// TwinCAT 3 PLC project HMI_Library
// Title: IBF_HMI
// Company: Industrial Brains B.V.
// ProjectVersion: 0.0.0.0
// Description: Basic HMI screens for use with Utilities and device libraries
// ProgramVersion: 3.1.4023.0
// libraries:
//   IBF_Device, * (Industrial Brains B.V.)
//   IBF_Utilities, * (Industrial Brains B.V.)
//   Tc2_Standard, * (Beckhoff Automation GmbH)
//   VisuDialogs, * (System)
//   VisuUserMgmt, * (System)
// project tree:
//   GVL/ E_BaseVisu.TcTLEO (not stored), GVL_HMI.TcGVL
//   HMIControl/ FB_HMIControl.TcPOU
//   IconsAndPictures/Backgrounds/PNG/ BackgroundImagePool_PNG.TcIPO (not stored)
//   IconsAndPictures/Backgrounds/SVG/ BackGroundImagePool_SVG.TcIPO (not stored)
//   IconsAndPictures/Buttons/ Buttons_SVG.TcIPO (not stored), Buttons_PNG.TcIPO (not stored)
//   IconsAndPictures/Logos/ LogoPool_PNG.TcIPO (not stored), LogoPool_SVG.TcIPO (not stored)
//   InputFunctions/ FB_HMILREALInput.TcPOU, FB_HMIInputBase.TcPOU
//   Screens/Backgrounds/ BackgroundNoButton.TcVIS, Background_SafetyAndSettings_SVG.TcVIS, BackgroundWithBorder.TcVIS
//   Screens/Base/ BaseScreen.TcVIS
//   Screens/EventsAndMessage/ BasicMessageScreen.TcVIS, Estop.TcVIS, MessageScreen.TcVIS (excluded from build)
//   Screens/Manual/DeviceScreens/ VisuAnalogOutControl.TcVIS, VisuAnalogAxisControl.TcVIS, VisuAnlogInputControl.TcVIS, VisuAxisControl.TcVIS, VisuCylinderControl.TcVIS, VisuDigitalInputControl.TcVIS, VisuDigitalOutControl.TcVIS, VisuEncoderInput.TcVIS, VisuKL5151Control.TcVIS, VisuKL15XXControl.TcVIS, VisuPushbuttonLightControl.TcVIS, VisuPWMControl.TcVIS, VisuDoublePWMControl.TcVIS, VisuUndefinedControl.TcVIS, VisuValveControl.TcVIS, VisuTwoVelocityAxisControl.TcVIS
//   Screens/Manual/ ManualButton_PNG.TcVIS, ManualControl.TcVIS, toManualButton.TcVIS
//   Screens/Parameter/ ParameterControl.TcVIS, ParButton_PNG.TcVIS
//   Screens/Startup Screen/ LogoScreen_PNG.TcVIS, LogoScreenBliss_PNG.TcVIS, LogoScreen_SVG.TcVIS, LogoScreenBlanc_SVG.TcVIS
//   Screens/State_PNG/ Idle_PNG.TcVIS, Manual_PNG.TcVIS, Parameter_PNG.TcVIS, Settings_PNG.TcVIS
//   Screens/State_SVG/ Manual.TcVIS, ParameterScreen.TcVIS, Settings.TcVIS, Idle.TcVIS
//   TextLists/ E_ComponentTypes.TcTLO, E_FaultTypes.TcTLO, E_Locations.TcTLO, E_MessageNumbers.TcTLO, E_ParameterNames.TcTLO, GlobalTextList.TcGTLO, TL_MessageDiscriptions.TcTLO
//   / VisualizationManager.TcVMO (not stored)

// ---- GVL/GVL_HMI.TcGVL
{attribute 'qualified_only'}
VAR_GLOBAL
	fbHMIControl	: FB_HMIControl ; // HMI control function
	bCmdSemiAuto	: BOOL ; // Show semi automatic screen
	bCmdAutomatic 	: BOOL ; // Show automatic screen
	eShownScreen 	: E_BaseVisu := E_BaseVisu.Idle ;
	bCmdSettings	: BOOL := FALSE ; // show settings screen
	bCmdParemeter	: BOOL := FALSE ; // Show paremeter screen
	bCmdManual		: BOOL := FALSE ; // Show manual screen
	bEstopActive	: BOOL ; // emergency stop is active
	sCmdEstopText	: STRING := 'SAFETY FAULT' ; // Emergency stop screen text 
	nStartVisu		: E_BaseVisu := E_BaseVisu.Idle ;
	nSelectedMessage : INT; 
END_VAR

// ---- HMIControl/FB_HMIControl.TcPOU
FUNCTION_BLOCK FB_HMIControl
VAR_INPUT 
END_VAR
VAR_OUTPUT
	bHideMessage	: BOOL ;
	bHideEStop 		: BOOL ;
	bHideBorders	: BOOL ;
	sEstopText		: STRING ;
	sOperatorMessage: STRING ;
END_VAR
VAR // HMI
END_VAR
VAR
	bWritePar  			: BOOL ; // write paremeters 
	bReadPar			: BOOL ; // Read paremeter file
	feWriteParemeter 	: F_TRIG ; // Falling edge trigger on leaving paremeter or manual screen

	reToSettings 		: R_TRIG ; // go to settings
	ePreviousScreen		: E_BaseVisu ; // previous screen
	
	bDisableSettings	: BOOL ; // disable settings button
END_VAR

SetScreen();
SetPopups();
ButtonEnable();

METHOD PRIVATE ButtonEnable : BOOL
VAR_INPUT
END_VAR
// Disable Buttons 
	bDisableSettings := GVL_HMI.eShownScreen = E_BaseVisu.Automatic ;
END_METHOD

METHOD PRIVATE SetPopups : BOOL
VAR_INPUT
END_VAR
// Set popup screens 
bHideEStop 			:= NOT GVL_HMI.bEstopActive ;
bHideMessage 		:= GVL_Message.bHideFaults ;
sOperatorMessage 	:= GVL_Message.sOPeratorMessage ;

GVL_HMI.bEstopActive := FALSE ;
END_METHOD

METHOD INTERNAL SetScreen : BOOL
VAR_INPUT
END_VAR
// Look for edges 
	reToSettings		( CLK := GVL_HMI.bCmdSettings );
	feWriteParemeter 	( CLK := GVL_HMI.bCmdParemeter OR GVL_HMI.bCmdManual );

// save previous screen 
IF reToSettings.Q  THEN 
	ePreviousScreen := GVL_HMI.eShownScreen ;
END_IF	
	
// Hide border control 
bHideBorders := FALSE ;

// Check active screen	
IF GVL_HMI.bCmdParemeter THEN 
	GVL_HMI.eShownScreen 	:= E_BaseVisu.Parameter ;
ELSIF GVL_HMI.bCmdManual THEN 
	GVL_HMI.eShownScreen 	:= E_BaseVisu.Manual;
ELSIF GVL_HMI.bCmdSettings THEN 
	GVL_HMI.eShownScreen 	:= E_BaseVisu.Settings ;
ELSIF NOT GVL_HMI.bCmdSettings AND GVL_HMI.eShownScreen = E_BaseVisu.Settings THEN 
	GVL_HMI.eShownScreen	:= ePreviousScreen ;
ELSIF gvl_HMI.bCmdSemiAuto THEN 
	GVL_HMI.eShownScreen 	:= E_BaseVisu.SemiAutomatic;
	gvl_HMI.bCmdSemiAuto	:= FALSE ; 
ELSIF gvl_HMI.bCmdAutomatic THEN 
	GVL_HMI.eShownScreen := E_BaseVisu.Automatic ;
	gvl_HMI.bCmdSemiAuto	:= FALSE ;
ELSE 
	GVL_HMI.eShownScreen := E_BaseVisu.Idle;
	bHideBorders := TRUE  ;	
END_IF

// Write parameters to file
IF feWriteParemeter.Q THEN
	bWritePar := TRUE ;
END_IF

IF bWritePar THEN 
	bWritePar R= GVL_Parameters.fbParameterHandler.CmdSavePar();
END_IF
END_METHOD

END_FUNCTION_BLOCK

// ---- InputFunctions/FB_HMILREALInput.TcPOU
FUNCTION_BLOCK PUBLIC FB_HMILREALInput EXTENDS FB_HMIInputBase // Analog value input from HMI
VAR_INPUT
	fInputFromHMI	: LREAL ;
END_VAR
VAR_OUTPUT
	fOutputToPLC	: LREAL ;
END_VAR
VAR
END_VAR

// call base function 
SUPER^();

// Set output to PLC
SetOutputToPLC();

METHOD PUBLIC SetOutputToPLC : BOOL
VAR_INPUT
END_VAR
IF bEnable THEN 
	fOutputToPLC := fInputFromHMI ;
END_IF
END_METHOD

END_FUNCTION_BLOCK

// ---- InputFunctions/FB_HMIInputBase.TcPOU
FUNCTION_BLOCK ABSTRACT FB_HMIInputBase //Base function for HMI inputs
VAR_INPUT
	bEnable : BOOL := TRUE ;
END_VAR
VAR_OUTPUT
	bInVisible			: BOOL := TRUE ; // input is visible (standard := NOT bEnable )
	bDeactivateInput	: BOOL := TRUE ; // input is enabled (Standard := bEnable)
END_VAR
VAR
END_VAR

SetHMIInstructions();

METHOD INTERNAL SetHMIInstructions : BOOL
VAR_INPUT
END_VAR
bInVisible 			:= NOT bEnable ;
bDeactivateInput	:= NOT bEnable ;
END_METHOD

METHOD ABSTRACT SetOutputToPLC : BOOL
VAR_INPUT
END_VAR
END_METHOD

END_FUNCTION_BLOCK

// ---- Screens/Backgrounds/BackgroundNoButton.TcVIS
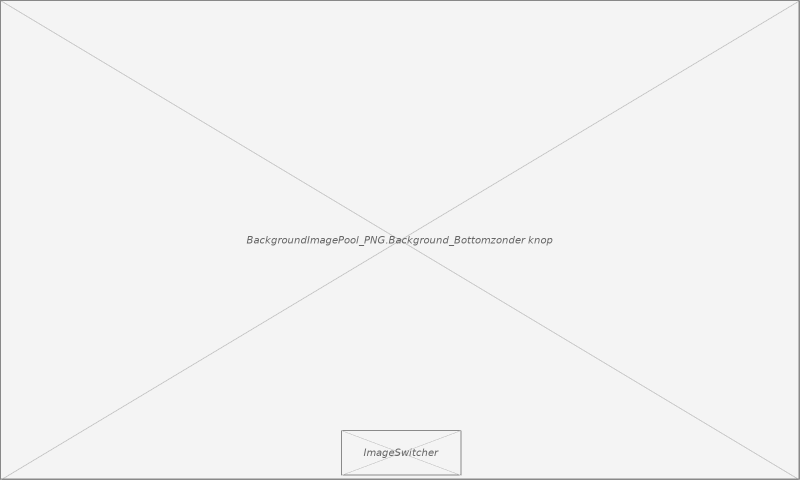
VISUALIZATION BackgroundNoButton  // 800x480
VAR_INPUT
	bHideEstop 			: BOOL ; // Hide emergency stop screen
	bDisableSettings	: BOOL ; // Deactivate settings
END_VAR
VAR_IN_OUT
	bCmdSettings	: BOOL ; // go to settings screen command
END_VAR
    Image (0,0 800x480), invisible if: bHideEstop, input disabled if: bHideEstop, image: BackgroundImagePool_PNG.Emergency Stop Active
    Image (0,0 800x480), image: BackgroundImagePool_PNG.Background_Bottomzonder knop
    ImageSwitcher (341,430 120x45), variable: GVL_HMI.bCmdSettings, input disabled if: bDisableSettings, background image: Buttons_PNG.Home-Settings Switch Pushed, image: Buttons_PNG.Home-Settings Switch, behaviour: TOGGLE
        p3148411668: Buttons_PNG.Home-Settings Switch Pushed
END_VISUALIZATION

// ---- Screens/Backgrounds/Background_SafetyAndSettings_SVG.TcVIS
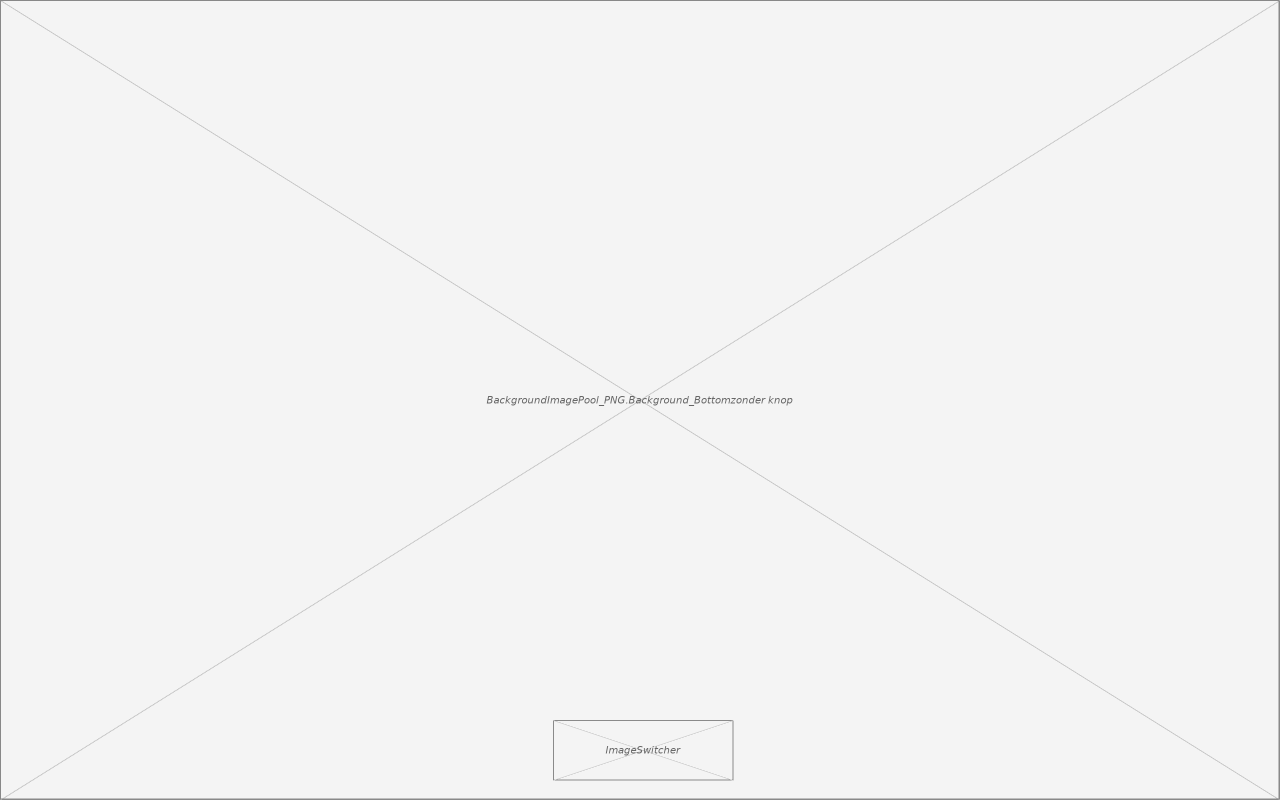
VISUALIZATION Background_SafetyAndSettings_SVG  // 1280x800
VAR_INPUT
	bHideEstop 			: BOOL ; // Hide emergency stop screen
	bDisableSettings	: BOOL ; // Deactivate settings
END_VAR
VAR_IN_OUT
	bCmdSettings	: BOOL ; // go to settings screen command
END_VAR
    Image (0,0 1280x800), invisible if: bHideEstop, input disabled if: bHideEstop, image: BackGroundImagePool_SVG.Emergency Stop Active 1280 x 800 Red Filled
    Image (0,0 1280x800), image: BackgroundImagePool_PNG.Background_Bottomzonder knop
    ImageSwitcher (553,720 180x60), variable: GVL_HMI.bCmdSettings, input disabled if: bDisableSettings, background image: Buttons_PNG.Home-Settings Switch Pushed, image: Buttons_PNG.Home-Settings Switch, behaviour: TOGGLE
        p3148411668: Buttons_PNG.Home-Settings Switch Pushed
END_VISUALIZATION

// ---- Screens/Backgrounds/BackgroundWithBorder.TcVIS
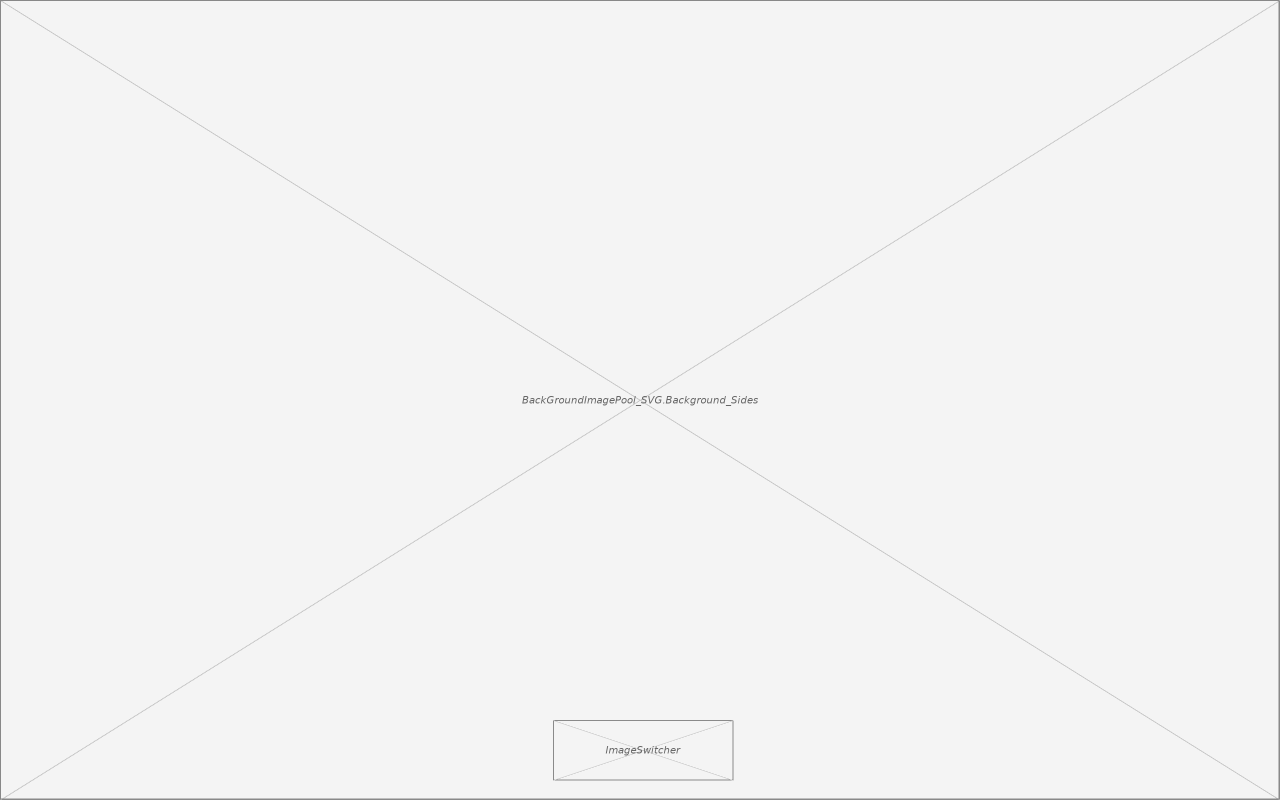
VISUALIZATION BackgroundWithBorder  // 1280x800
    Image (0,710 1280x90), image: BackGroundImagePool_SVG.Background_Bottom
    Image (0,0 1280x800), invisible if: GVL_HMI.fbHMIControl.bHideBorders, image: BackGroundImagePool_SVG.Background_Sides
    ImageSwitcher (553,720 180x60), variable: GVL_HMI.bCmdSettings, input disabled if: GVL_HMI.fbHMIControl.bDisableSettings, background image: Buttons_SVG.Home-Settings Switch Pushed, image: Buttons_SVG.Home Settings switch, behaviour: TOGGLE
        p3148411668: Buttons_SVG.Home-Settings Switch Pushed
END_VISUALIZATION

// ---- Screens/Base/BaseScreen.TcVIS
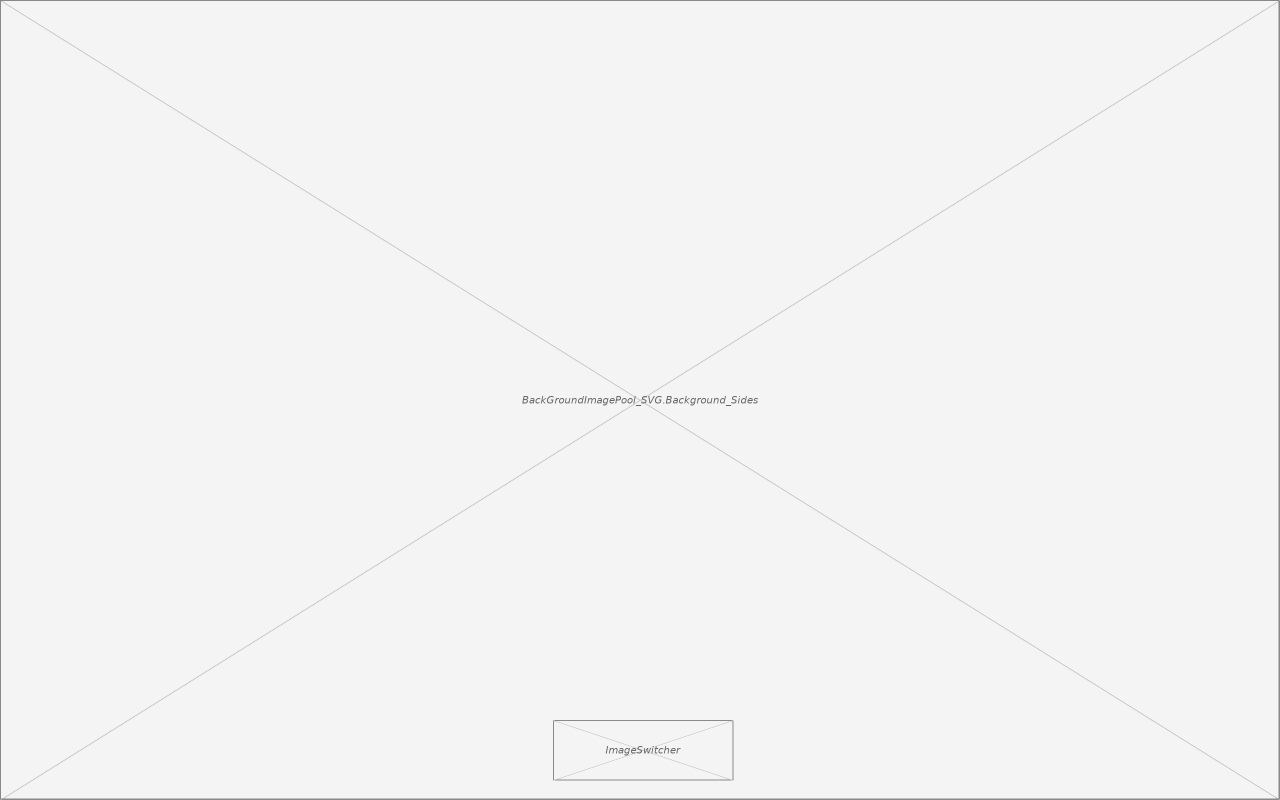
VISUALIZATION BaseScreen  // 1280x800
    Frame (0,0 1280x800)
        shows BackgroundWithBorder()
END_VISUALIZATION

// ---- Screens/EventsAndMessage/BasicMessageScreen.TcVIS
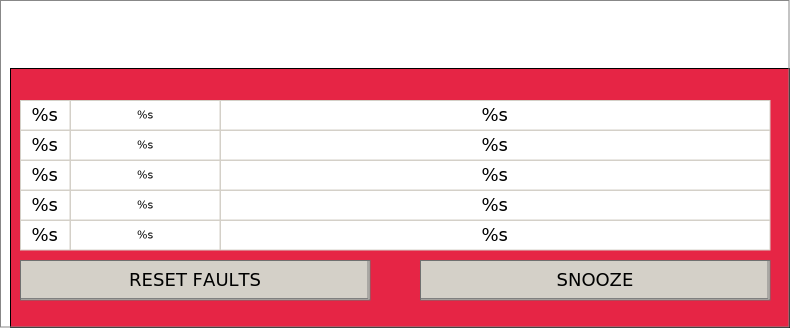
VISUALIZATION BasicMessageScreen  // 790x328
    RoundedRectangle (10,68 780x260)
    Group (20,100 754x200), invisible if: Utilities_Library.GVL_Message.bHideFaults, input disabled if: Utilities_Library.GVL_Message.bHideFaults
        Group (0,0 750x30)
            Textfield (0,0 50x30), "%s", text variable: GVL_Message.arActiveFaults[0].FaultType
            Textfield (50,0 150x30), "%s", text variable: Utilities_Library.GVL_Message.arActiveFaults[0].FullFaultId
            Textfield (200,0 550x30), "%s", text variable: Utilities_Library.GVL_Message.arActiveFaults[0].Discription
        Group (0,30 750x30)
            Textfield (0,0 50x30), "%s", text variable: Utilities_Library.GVL_Message.arActiveFaults[1].FaultType
            Textfield (50,0 150x30), "%s", text variable: Utilities_Library.GVL_Message.arActiveFaults[1].FullFaultId
            Textfield (200,0 550x30), "%s", text variable: Utilities_Library.GVL_Message.arActiveFaults[1].Discription
        Group (0,60 750x30)
            Textfield (0,0 50x30), "%s", text variable: Utilities_Library.GVL_Message.arActiveFaults[2].FaultType
            Textfield (50,0 150x30), "%s", text variable: Utilities_Library.GVL_Message.arActiveFaults[2].FullFaultId
            Textfield (200,0 550x30), "%s", text variable: Utilities_Library.GVL_Message.arActiveFaults[2].Discription
        Group (0,90 750x30)
            Textfield (0,0 50x30), "%s", text variable: Utilities_Library.GVL_Message.arActiveFaults[3].FaultType
            Textfield (50,0 150x30), "%s", text variable: Utilities_Library.GVL_Message.arActiveFaults[3].FullFaultId
            Textfield (200,0 550x30), "%s", text variable: Utilities_Library.GVL_Message.arActiveFaults[3].Discription
        Group (0,120 750x30)
            Textfield (0,0 50x30), "%s", text variable: Utilities_Library.GVL_Message.arActiveFaults[4].FaultType
            Textfield (50,0 150x30), "%s", text variable: Utilities_Library.GVL_Message.arActiveFaults[4].FullFaultId
            Textfield (200,0 550x30), "%s", text variable: Utilities_Library.GVL_Message.arActiveFaults[4].Discription
        Button (0,160 350x40), "RESET FAULTS", invisible if: Utilities_Library.GVL_Message.bHideReset, input disabled if: Utilities_Library.GVL_Message.bHideReset
            tap Utilities_Library.GVL_Message.bResetFaults
        Button (400,160 350x40), "SNOOZE"
            tap Utilities_Library.GVL_Message.bCmdSnoozeMessage
END_VISUALIZATION

// ---- Screens/EventsAndMessage/Estop.TcVIS
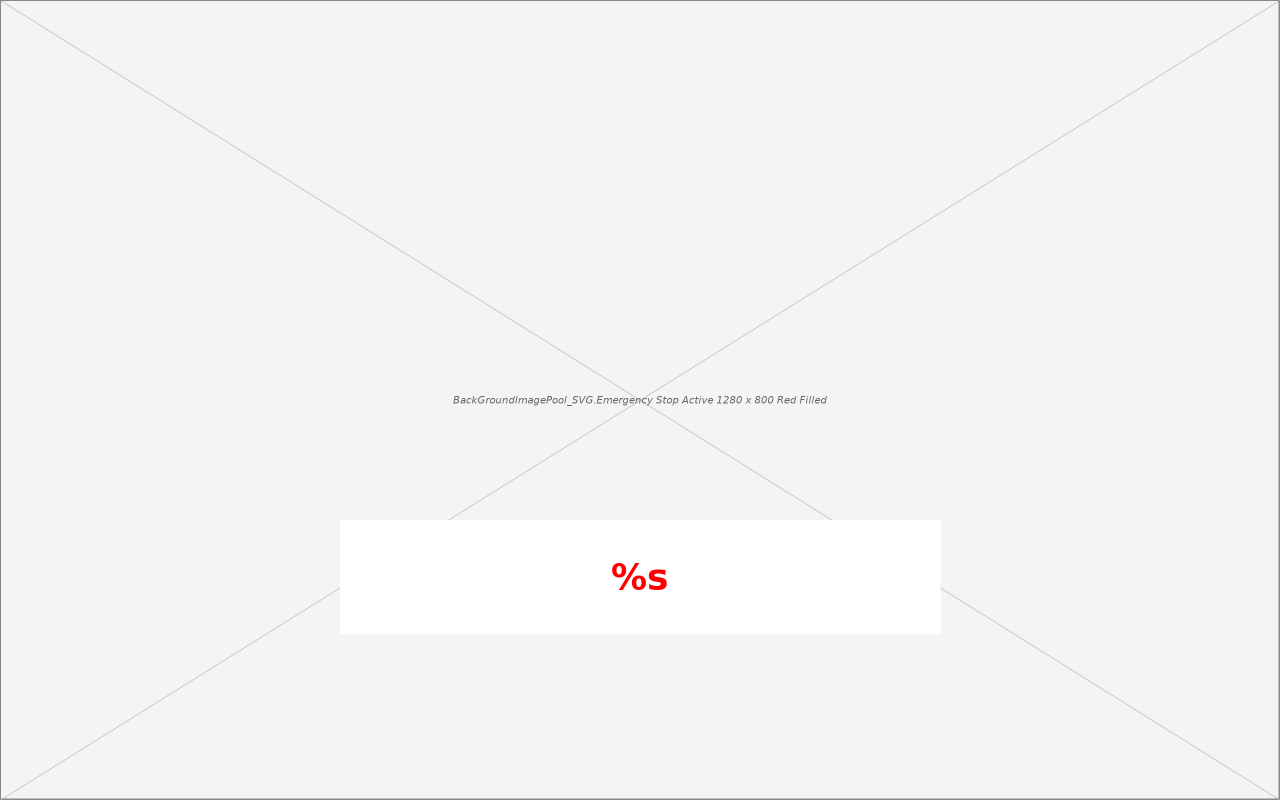
VISUALIZATION Estop  // 1280x800
VAR_IN_OUT
	bHideEstop		: BOOL ; // Hide Estop screen
END_VAR
    Image (0,0 1280x800), image: BackGroundImagePool_SVG.Emergency Stop Active 1280 x 800 Red Filled
    Textfield (340,520 600x114), "%s", text variable: GVL_HMI.sCmdEstopText
END_VISUALIZATION

// ---- Screens/Manual/DeviceScreens/VisuAnalogOutControl.TcVIS
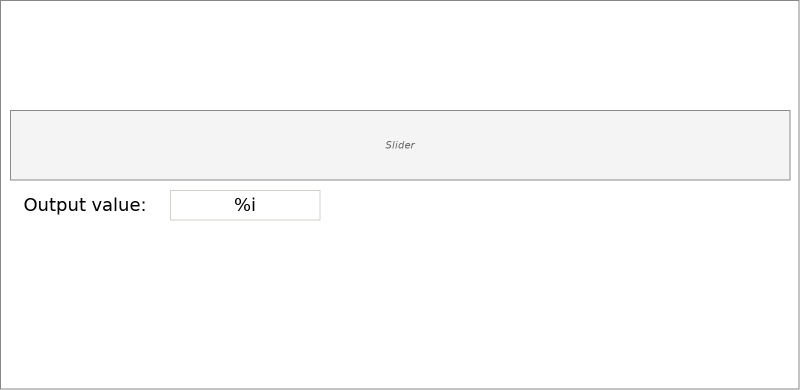
VISUALIZATION VisuAnalogOutControl  // 800x390
VAR_IN_OUT
	fbManualControler	: FB_ManualController ;
END_VAR
    Slider (10,110 780x70), variable: fbManualControler.pDevAnalogOut^.fCmdValue, scale 0..100
    Textfield (170,190 150x30), "%i", text variable: fbManualControler.pDevAnalogOut^.fCmdValue
        OnMouseClick: write the text variable via VisuDialogs.Numpad
    Label (10,190 150x30), "Output value:"
END_VISUALIZATION

// ---- Screens/Manual/DeviceScreens/VisuAnalogAxisControl.TcVIS
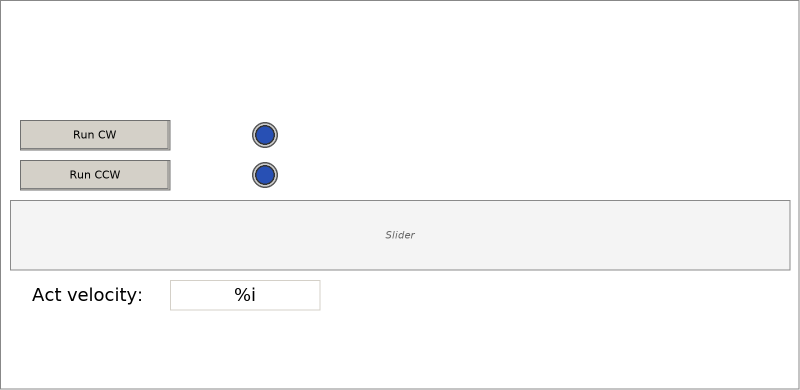
VISUALIZATION VisuAnalogAxisControl  // 800x390
VAR_IN_OUT
	fbManualControler	: FB_ManualController ;
END_VAR
    Slider (10,200 780x70), variable: fbManualControler.pDevAnalogAxis^.stManualCtrl.fCmdVelocity, scale 0..100
    Textfield (170,280 150x30), "%i", text variable: fbManualControler.pDevAnalogAxis^.fActVelocity
        OnMouseClick: write the text variable via VisuDialogs.Numpad
    Label (10,280 150x30), "Act velocity:"
    Button (20,120 150x30), "Run CW"
        tap fbManualControler.pDevAnalogAxis^.stManualCtrl.bCmdRunCW
    Button (20,160 150x30), "Run CCW"
        tap fbManualControler.pDevAnalogAxis^.stManualCtrl.bCmdRunCCW
    Lamp1 (190,120 150x30), variable: fbManualControler.pDevAnalogAxis^.bMovingCW, style: Lamp-Lamp1-Blue
    Lamp1 (190,160 150x30), variable: fbManualControler.pDevAnalogAxis^.bMovingCCW, style: Lamp-Lamp1-Blue
END_VISUALIZATION

// ---- Screens/Manual/DeviceScreens/VisuAnlogInputControl.TcVIS
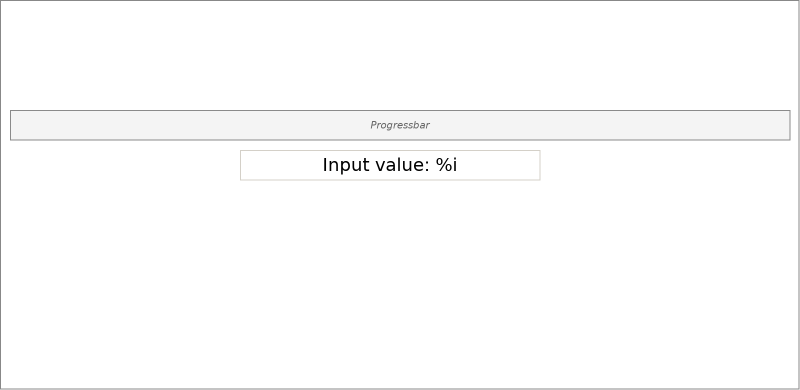
VISUALIZATION VisuAnlogInputControl  // 800x390
VAR_IN_OUT
	fbManualControler	: FB_ManualController ;
END_VAR
    Progressbar (10,110 780x30), variable: fbManualControler.pDevAnalogInput^.fValue
    Textfield (240,150 300x30), "Input value: %i", text variable: fbManualControler.pDevAnalogInput^.fValue
END_VISUALIZATION

// ---- Screens/Manual/DeviceScreens/VisuAxisControl.TcVIS
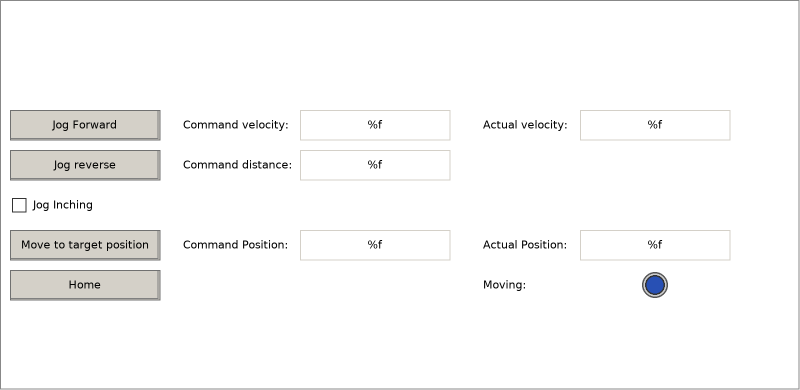
VISUALIZATION VisuAxisControl  // 800x390
VAR_IN_OUT
	fbManualControler	: FB_ManualController ;
END_VAR
    Button (10,110 150x30), "Jog Forward"
        tap fbManualControler.pDevAxis^.stManualCtrl.bCmdJogForward
    Button (10,150 150x30), "Jog reverse"
        tap fbManualControler.pDevAxis^.stManualCtrl.bCmdJogReverse
    Button (10,230 150x30), "Move to target position"
        tap fbManualControler.pDevAxis^.stManualCtrl.bCmdToPos
    Button (10,270 150x30), "Home"
        tap fbManualControler.pDevAxis^.stManualCtrl.bCmdHome
    Checkbox (10,190 150x30), "Jog Inching", variable: fbManualControler.pDevAxis^.stManualCtrl.bCmdInching
    Label (180,150 120x30), "Command distance:"
    Label (180,110 120x30), "Command velocity:"
    Label (180,230 120x30), "Command Position:"
    Textfield (300,110 150x30), "%f", text variable: fbManualControler.pDevAxis^.stManualCtrl.fVelocity
        OnMouseDown: write the text variable via VisuDialogs.Numpad
    Textfield (300,150 150x30), "%f", text variable: fbManualControler.pDevAxis^.stManualCtrl.fDistance
        OnMouseDown: write the text variable via VisuDialogs.Numpad
    Textfield (300,230 150x30), "%f", text variable: fbManualControler.pDevAxis^.stManualCtrl.fPosition
        OnMouseDown: write the text variable via VisuDialogs.Numpad
    Label (480,110 100x30), "Actual velocity:"
    Label (480,230 100x30), "Actual Position:"
    Textfield (580,230 150x30), "%f", text variable: fbManualControler.pDevAxis^.fActPosition
        OnMouseDown: write the text variable via VisuDialogs.Numpad
    Textfield (580,110 150x30), "%f", text variable: fbManualControler.pDevAxis^.fVelocity
        OnMouseDown: write the text variable via VisuDialogs.Numpad
    Lamp1 (580,270 150x30), variable: fbManualControler.pDevAxis^.AxisRef.Status.Moving, style: Lamp-Lamp1-Blue
    Label (480,270 100x30), "Moving:"
END_VISUALIZATION

// ---- Screens/Manual/DeviceScreens/VisuCylinderControl.TcVIS
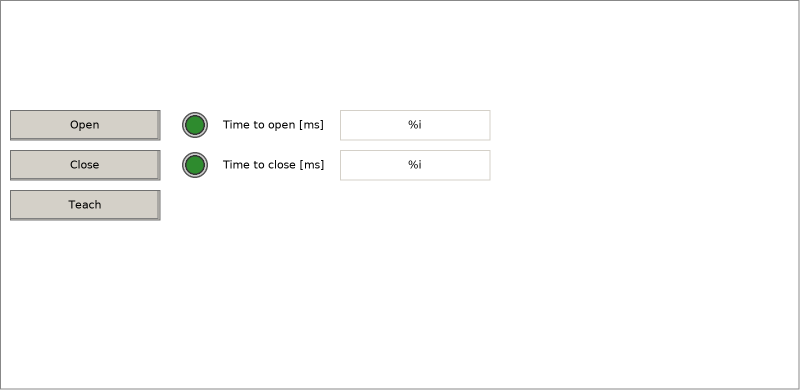
VISUALIZATION VisuCylinderControl  // 800x390
VAR_IN_OUT
	fbManualControler	: FB_ManualController ;
END_VAR
    Button (10,110 150x30), "Open"
        tap fbManualControler.pDevCylinder^.stManualCtrl.bCmdOpen
    Button (10,150 150x30), "Close"
        tap fbManualControler.pDevCylinder^.stManualCtrl.bCmdClose
    Lamp1 (180,110 30x30), variable: fbManualControler.pDevCylinder^.bFco_Open, style: Lamp-Lamp1-Green
    Button (10,190 150x30), "Teach"
        toggle fbManualControler.pDevCylinder^.stManualCtrl.bCmdTeach
    Lamp1 (180,150 30x30), variable: fbManualControler.pDevCylinder^.bFco_Closed, style: Lamp-Lamp1-Green
    Label (220,110 100x30), "Time to open [ms]"
    Label (220,150 100x30), "Time to close [ms]"
    Textfield (340,150 150x30), "%i", text variable: fbManualControler.pDevCylinder^.stParTimeToClose.fValue
        OnMouseClick: write the text variable via VisuDialogs.Numpad, min 0
    Textfield (340,110 150x30), "%i", text variable: fbManualControler.pDevCylinder^.stParTimeToOpen.fValue
        OnMouseClick: write the text variable via VisuDialogs.Numpad, min 0
END_VISUALIZATION

// ---- Screens/Manual/DeviceScreens/VisuDigitalInputControl.TcVIS
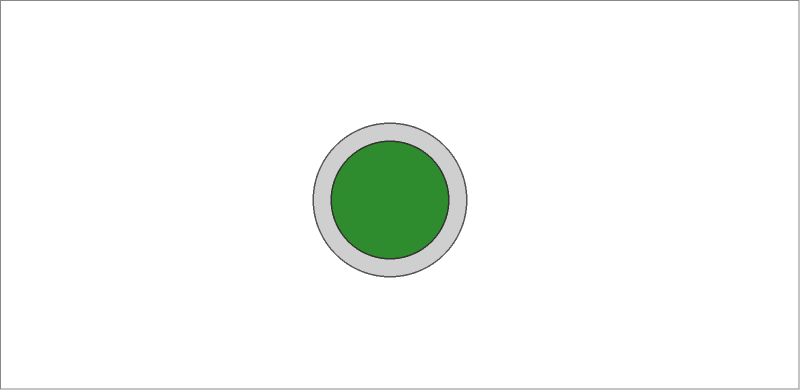
VISUALIZATION VisuDigitalInputControl  // 800x390
VAR_IN_OUT
	fbManualControler	: FB_ManualController ;
END_VAR
    Lamp1 (300,110 180x180), variable: fbManualControler.pDevDigitalInput^.bFcoInputActive, style: Lamp-Lamp1-Green
END_VISUALIZATION

// ---- Screens/Manual/DeviceScreens/VisuDigitalOutControl.TcVIS
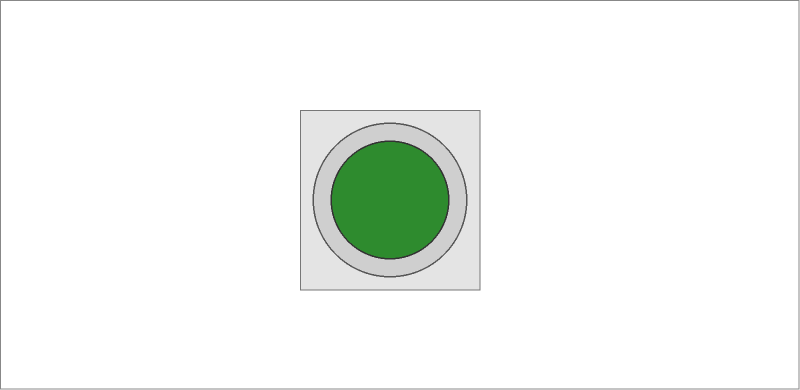
VISUALIZATION VisuDigitalOutControl  // 800x390
VAR_IN_OUT
	fbManualControler	: FB_ManualController ;
END_VAR
    PushSwitch (300,110 180x180), variable: fbManualControler.pDevDigitalOut^.bCmdOn, behaviour: TOGGLE, style: Switch-PushSwitch-Green
END_VISUALIZATION

// ---- Screens/Manual/DeviceScreens/VisuEncoderInput.TcVIS
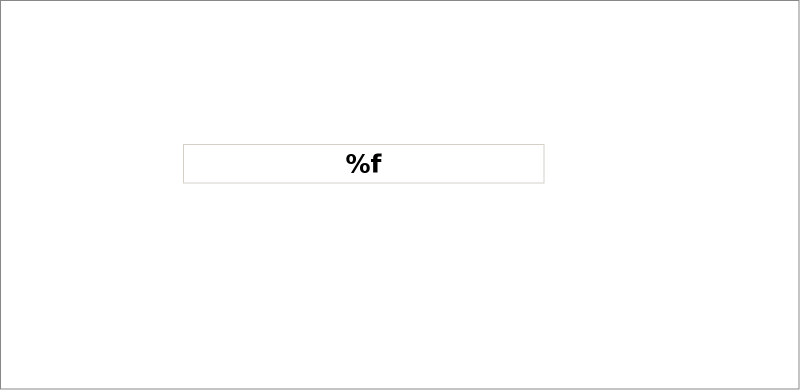
VISUALIZATION VisuEncoderInput  // 800x390
VAR_IN_OUT
	fbManualControler	: FB_ManualController ;
END_VAR
    Textfield (183,144 361x39), "%f", text variable: fbManualControler.pDevEncoder^.nOutPosition
END_VISUALIZATION

// ---- Screens/Manual/DeviceScreens/VisuKL5151Control.TcVIS
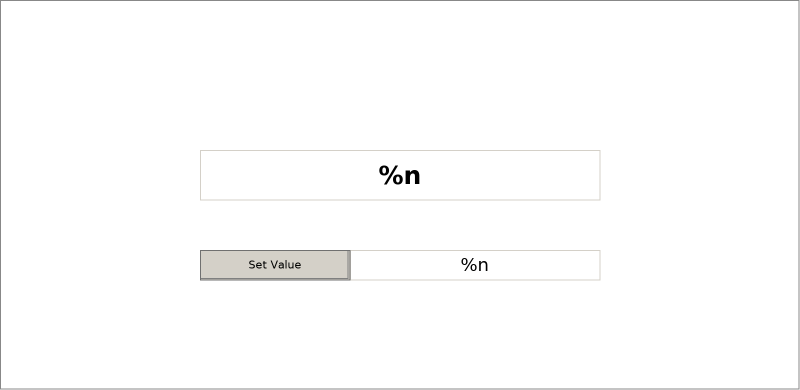
VISUALIZATION VisuKL5151Control  // 800x390
VAR_IN_OUT
	fbManualControler	: FB_ManualController ;
END_VAR
    Textfield (200,150 400x50), "%n", text variable: fbManualControler.pDevKL5151^.CountValue
    Textfield (350,250 250x30), "%n", text variable: fbManualControler.pDevKL5151^.stManualControl.nManValue
        OnMouseClick: write the text variable via VisuDialogs.Numpad
    Button (200,250 150x30), "Set Value"
        tap fbManualControler.pDevKL5151^.stManualControl.bManSetValue
END_VISUALIZATION

// ---- Screens/Manual/DeviceScreens/VisuKL15XXControl.TcVIS
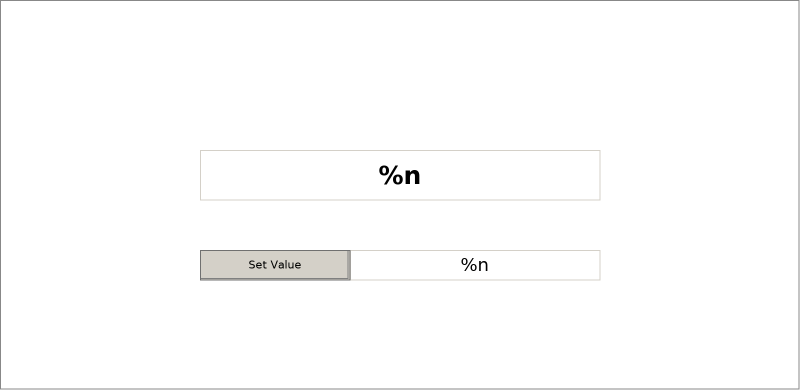
VISUALIZATION VisuKL15XXControl  // 800x390
VAR_IN_OUT
	fbManualControler	: FB_ManualController ;
END_VAR
    Textfield (200,150 400x50), "%n", text variable: fbManualControler.pDevKL1512^.CountValue
    Textfield (350,250 250x30), "%n", text variable: fbManualControler.pDevKL1512^.stManualControl.nManValue
        OnMouseClick: write the text variable via VisuDialogs.Numpad
    Button (200,250 150x30), "Set Value"
        tap fbManualControler.pDevKL1512^.stManualControl.bManSetValue
END_VISUALIZATION

// ---- Screens/Manual/DeviceScreens/VisuPushbuttonLightControl.TcVIS
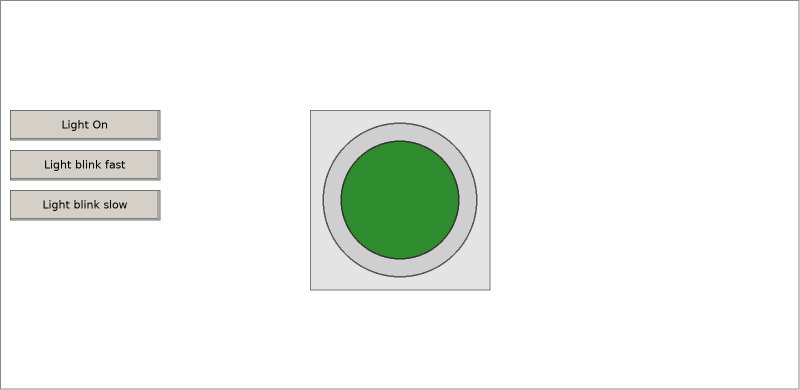
VISUALIZATION VisuPushbuttonLightControl  // 800x390
VAR_IN_OUT
	fbManualControler	: FB_ManualController ;
END_VAR
    PushSwitch (310,110 180x180), variable: fbManualControler.pDevPBL^.bFcoInputActive, behaviour: TOGGLE, style: Switch-PushSwitch-Green
    Button (10,110 150x30), "Light On"
        toggle fbManualControler.pDevPBL^.fbLight.bCmdOn
    Button (10,150 150x30), "Light blink fast"
        toggle fbManualControler.pDevPBL^.fbLight.bCmdBlinkFast
    Button (10,190 150x30), "Light blink slow"
        toggle fbManualControler.pDevPBL^.fbLight.bCmdBlinkSlow
END_VISUALIZATION

// ---- Screens/Manual/DeviceScreens/VisuPWMControl.TcVIS
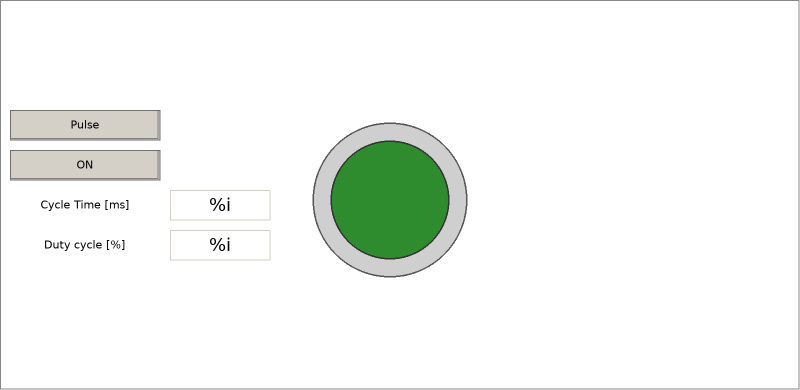
VISUALIZATION VisuPWMControl  // 800x390
VAR_IN_OUT
	fbManualControler	: FB_ManualController ;
END_VAR
    Lamp1 (300,110 180x180), variable: fbManualControler.pDevPWMController^.qbOutput, style: Lamp-Lamp1-Green
    Button (10,110 150x30), "Pulse"
        toggle fbManualControler.pDevPWMController^.bCmdPWMCycle
    Button (10,150 150x30), "ON"
        tap fbManualControler.pDevPWMController^.bCmdOn
    Textfield (170,190 100x30), "%i", text variable: fbManualControler.pDevPWMController^.nPeriodLength
        OnMouseUp: write the text variable via VisuDialogs.Numpad
    Label (10,190 150x30), "Cycle Time [ms]"
    Label (10,230 150x30), "Duty cycle [%]"
    Textfield (170,230 100x30), "%i", text variable: fbManualControler.pDevPWMController^.nDutyCycle
        OnMouseClick: write the text variable via VisuDialogs.Numpad, min 0, max 100
END_VISUALIZATION

// ---- Screens/Manual/DeviceScreens/VisuDoublePWMControl.TcVIS
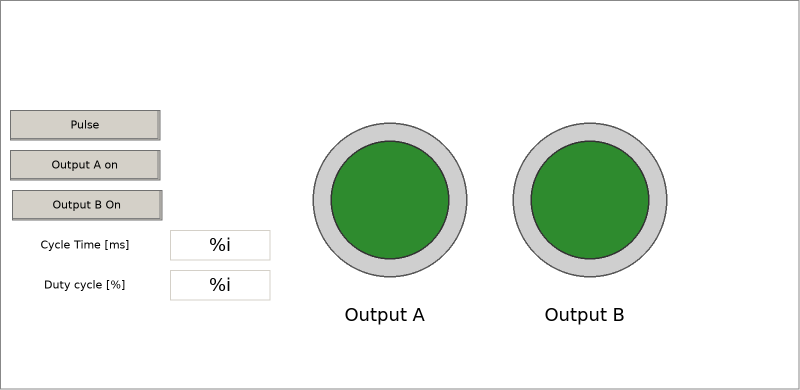
VISUALIZATION VisuDoublePWMControl  // 800x390
VAR_IN_OUT
	fbManualControler	: FB_ManualController ;
END_VAR
    Lamp1 (300,110 180x180), variable: fbManualControler.pDevDoublePWM^.qbOutputA, style: Lamp-Lamp1-Green
    Button (10,110 150x30), "Pulse"
        toggle fbManualControler.pDevDoublePWM^.bCmdPWMOn
    Button (10,150 150x30), "Output A on"
        toggle fbManualControler.pDevDoublePWM^.bCmdChanelAOn
    Textfield (170,230 100x30), "%i", text variable: fbManualControler.pDevDoublePWM^.stParPeriodLength.fValue
        OnMouseUp: write the text variable via VisuDialogs.Numpad
    Label (10,230 150x30), "Cycle Time [ms]"
    Label (10,270 150x30), "Duty cycle [%]"
    Textfield (170,270 100x30), "%i", text variable: fbManualControler.pDevDoublePWM^.stParDutyCycle.fValue
        OnMouseClick: write the text variable via VisuDialogs.Numpad, min 0, max 100
    Lamp1 (500,110 180x180), variable: fbManualControler.pDevPWMController^.qbOutput, style: Lamp-Lamp1-Green
    Button (12,190 150x30), "Output B On"
        tap fbManualControler.pDevDoublePWM^.bCmdChanelBOn
    Label (310,300 150x30), "Output A"
    Label (510,300 150x30), "Output B"
END_VISUALIZATION

// ---- Screens/Manual/DeviceScreens/VisuUndefinedControl.TcVIS
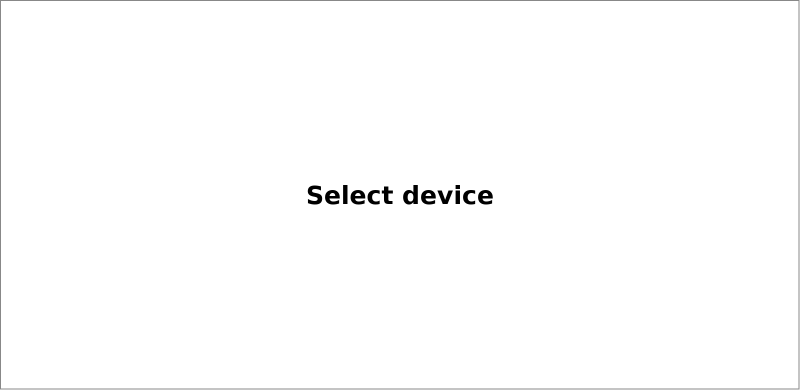
VISUALIZATION VisuUndefinedControl  // 800x390
    Label (0,0 800x390), "Select device"
END_VISUALIZATION

// ---- Screens/Manual/DeviceScreens/VisuValveControl.TcVIS
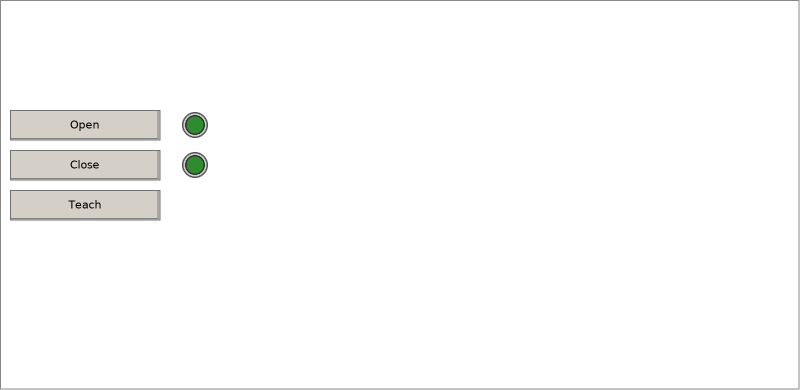
VISUALIZATION VisuValveControl  // 800x390
VAR_IN_OUT
	fbManualControler	: FB_ManualController ;
END_VAR
    Button (10,110 150x30), "Open"
        tap fbManualControler.pDevValve^.stManualCtrl.bCmdOpen
    Button (10,150 150x30), "Close"
        tap fbManualControler.pDevValve^.stManualCtrl.bCmdClose
    Lamp1 (180,110 30x30), variable: fbManualControler.pDevValve^.bFco_Open, style: Lamp-Lamp1-Green
    Button (10,190 150x30), "Teach"
        toggle fbManualControler.pDevValve^.stManualCtrl.bCmdTeach
    Lamp1 (180,150 30x30), variable: fbManualControler.pDevValve^.bFco_Closed, style: Lamp-Lamp1-Green
END_VISUALIZATION

// ---- Screens/EventsAndMessage/MessageScreen.TcVIS
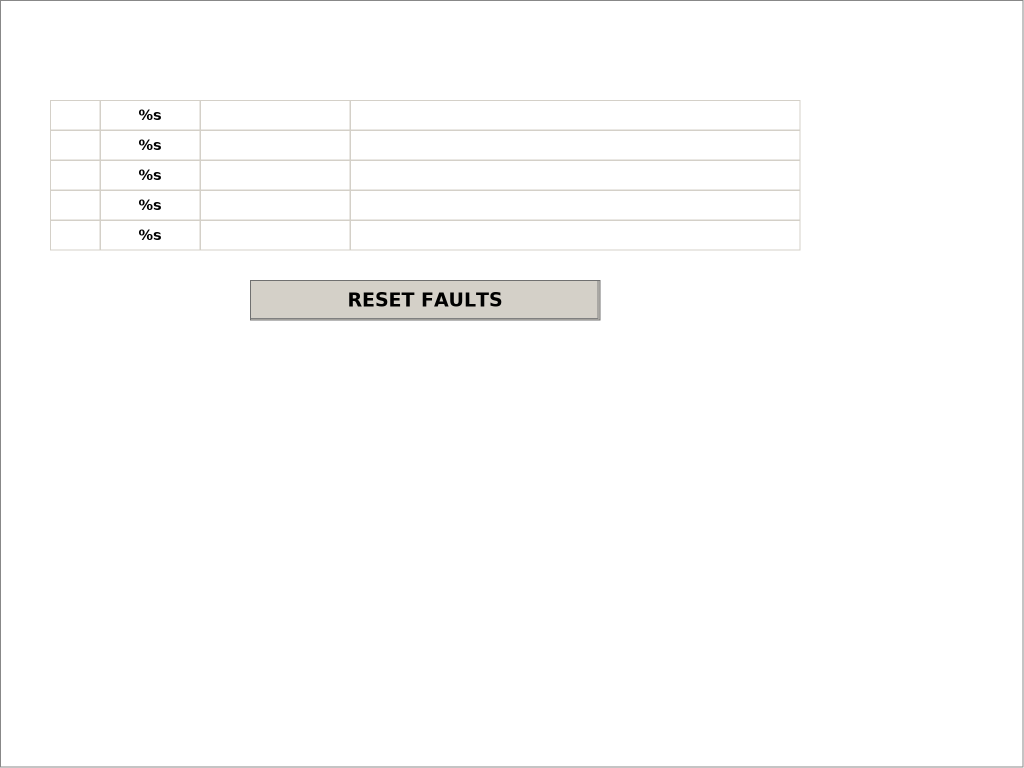
VISUALIZATION MessageScreen  // 1024x768
    Group (50,100 750x220)
        Group (0,0 750x30)
            Textfield (0,0 50x30), text list: 'E_FaultTypes', text index: Utilities_Library.GVL_Message.arActiveFaults[0].FaultType
            Textfield (50,0 100x30), "%s", text variable: Utilities_Library.GVL_Message.arActiveFaults[0].FullFaultId
            Textfield (150,0 150x30), text list: 'E_Locations', text index: Utilities_Library.GVL_Message.arActiveFaults[0].LocationNumber
            Textfield (300,0 450x30), text list: 'TL_MessageDiscriptions', text index: Utilities_Library.GVL_Message.arActiveFaults[0].MessageNumber
        Group (0,30 750x30)
            Textfield (0,0 50x30), text list: 'E_FaultTypes', text index: Utilities_Library.GVL_Message.arActiveFaults[1].FaultType
            Textfield (50,0 100x30), "%s", text variable: Utilities_Library.GVL_Message.arActiveFaults[1].FullFaultId
            Textfield (150,0 150x30), text list: 'E_Locations', text index: Utilities_Library.GVL_Message.arActiveFaults[1].LocationNumber
            Textfield (300,0 450x30), text list: 'TL_MessageDiscriptions', text index: Utilities_Library.GVL_Message.arActiveFaults[1].MessageNumber
        Group (0,60 750x30)
            Textfield (0,0 50x30), text list: 'E_FaultTypes', text index: Utilities_Library.GVL_Message.arActiveFaults[2].FaultType
            Textfield (50,0 100x30), "%s", text variable: Utilities_Library.GVL_Message.arActiveFaults[2].FullFaultId
            Textfield (150,0 150x30), text list: 'E_Locations', text index: Utilities_Library.GVL_Message.arActiveFaults[2].LocationNumber
            Textfield (300,0 450x30), text list: 'TL_MessageDiscriptions', text index: Utilities_Library.GVL_Message.arActiveFaults[2].MessageNumber
        Group (0,90 750x30)
            Textfield (0,0 50x30), text list: 'E_FaultTypes', text index: Utilities_Library.GVL_Message.arActiveFaults[3].FaultType
            Textfield (50,0 100x30), "%s", text variable: Utilities_Library.GVL_Message.arActiveFaults[3].FullFaultId
            Textfield (150,0 150x30), text list: 'E_Locations', text index: Utilities_Library.GVL_Message.arActiveFaults[3].LocationNumber
            Textfield (300,0 450x30), text list: 'TL_MessageDiscriptions', text index: Utilities_Library.GVL_Message.arActiveFaults[3].MessageNumber
        Group (0,120 750x30)
            Textfield (0,0 50x30), text list: 'E_FaultTypes', text index: Utilities_Library.GVL_Message.arActiveFaults[4].FaultType
            Textfield (50,0 100x30), "%s", text variable: Utilities_Library.GVL_Message.arActiveFaults[4].FullFaultId
            Textfield (150,0 150x30), text list: 'E_Locations', text index: Utilities_Library.GVL_Message.arActiveFaults[4].LocationNumber
            Textfield (300,0 450x30), text list: 'TL_MessageDiscriptions', text index: Utilities_Library.GVL_Message.arActiveFaults[4].MessageNumber
        Button (200,180 350x40), "RESET FAULTS"
            tap Utilities_Library.GVL_Message.bResetFaults
END_VISUALIZATION

// ---- Screens/Manual/DeviceScreens/VisuTwoVelocityAxisControl.TcVIS
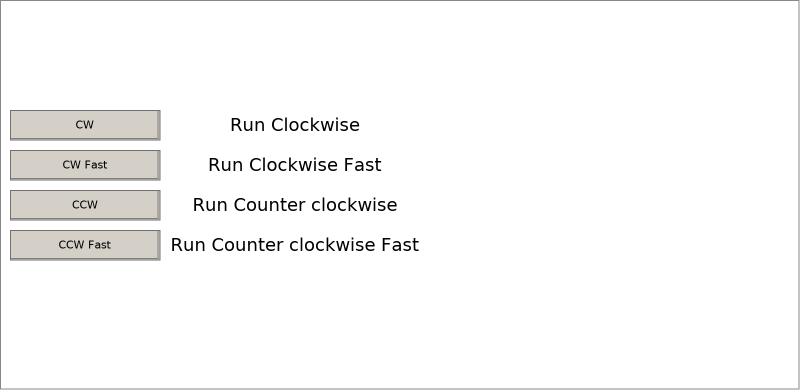
VISUALIZATION VisuTwoVelocityAxisControl  // 800x390
VAR_IN_OUT
	fbManualControler	: FB_ManualController ;
END_VAR
    Button (10,110 150x30), "CW"
        tap fbManualControler.pDevTwoVelocityAxis^.stManualControl.bManRunCW
    Button (10,150 150x30), "CW Fast"
        tap fbManualControler.pDevTwoVelocityAxis^.stManualControl.bManRunCWFast
    Button (10,190 150x30), "CCW"
        tap fbManualControler.pDevTwoVelocityAxis^.stManualControl.bManRunCCw
    Button (10,230 150x30), "CCW Fast"
        tap fbManualControler.pDevTwoVelocityAxis^.stManualControl.bManRunCCWFast
    Label (170,110 250x30), "Run Clockwise"
    Label (170,150 250x30), "Run Clockwise Fast"
    Label (170,190 250x30), "Run Counter clockwise"
    Label (170,230 250x30), "Run Counter clockwise Fast"
END_VISUALIZATION

// ---- Screens/Manual/ManualButton_PNG.TcVIS
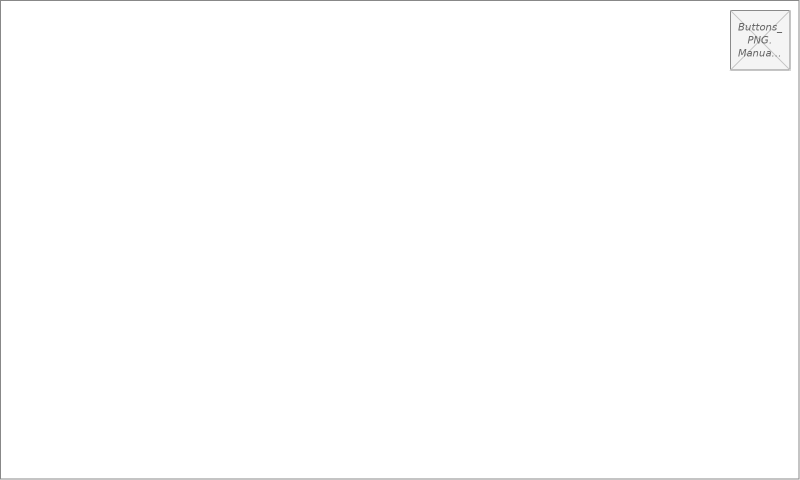
VISUALIZATION ManualButton_PNG  // 800x480
VAR_IN_OUT
	bCmdManual	: BOOL ; // switch to manual screen
END_VAR
    Image (730,10 60x60), image: Buttons_PNG.Manual mode Idle
        OnMouseClick: VisuUserMgmt Type=Login
        OnMouseClick: toggle bCmdManual
END_VISUALIZATION

// ---- Screens/Manual/ManualControl.TcVIS
